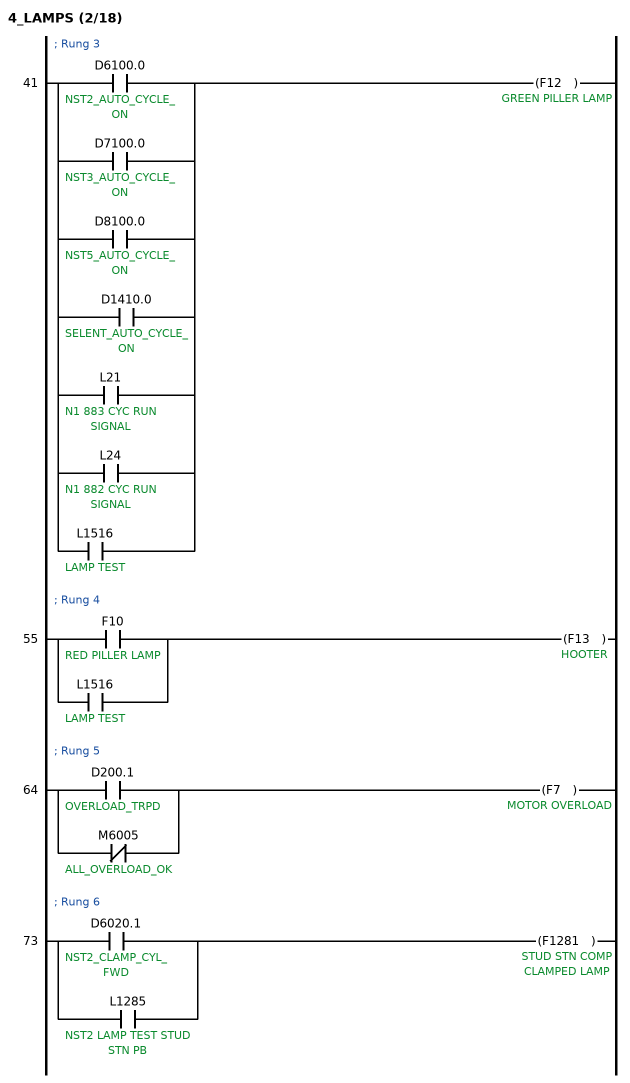
[picture p48: ladder of 4_LAMPS, rungs at steps 41 to 73]
; Rung 3
41    LD      D6100.0  ; NST2_AUTO_CYCLE_ON
      OR      D7100.0  ; NST3_AUTO_CYCLE_ON
      OR      D8100.0  ; NST5_AUTO_CYCLE_ON
      OR      D1410.0  ; SELENT_AUTO_CYCLE_ON
      OR      L21  ; N1 883 CYC RUN SIGNAL
      OR      L24  ; N1 882 CYC RUN SIGNAL
      OR      L1516  ; LAMP TEST
      OUT     F12  ; GREEN PILLER LAMP
; Rung 4
55    LD      F10  ; RED PILLER LAMP
      OR      L1516  ; LAMP TEST
      OUT     F13  ; HOOTER
; Rung 5
64    LD      D200.1  ; OVERLOAD_TRPD
      ORI     M6005  ; ALL_OVERLOAD_OK
      OUT     F7  ; MOTOR OVERLOAD
; Rung 6
73    LD      D6020.1  ; NST2_CLAMP_CYL_FWD
      OR      L1285  ; NST2 LAMP TEST STUD STN PB
      OUT     F1281  ; STUD STN COMP CLAMPED LAMP
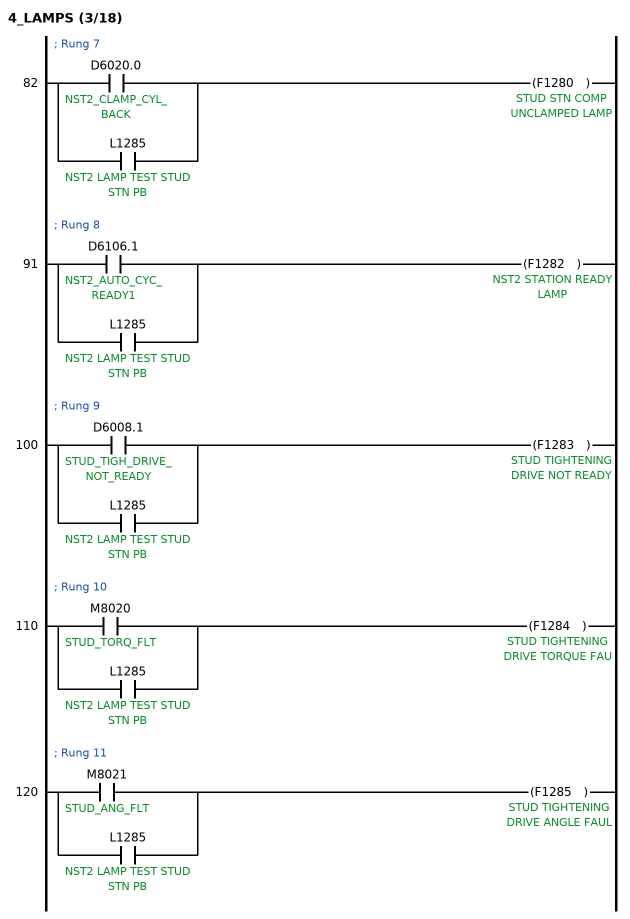
; Rung 7
82    LD      D6020.0  ; NST2_CLAMP_CYL_BACK
      OR      L1285  ; NST2 LAMP TEST STUD STN PB
      OUT     F1280  ; STUD STN COMP UNCLAMPED LAMP
; Rung 8
91    LD      D6106.1  ; NST2_AUTO_CYC_READY1
      OR      L1285  ; NST2 LAMP TEST STUD STN PB
      OUT     F1282  ; NST2 STATION READY LAMP
; Rung 9
100   LD      D6008.1  ; STUD_TIGH_DRIVE_NOT_READY
      OR      L1285  ; NST2 LAMP TEST STUD STN PB
      OUT     F1283  ; STUD TIGHTENING DRIVE NOT READY
; Rung 10
110   LD      M8020  ; STUD_TORQ_FLT
      OR      L1285  ; NST2 LAMP TEST STUD STN PB
      OUT     F1284  ; STUD TIGHTENING DRIVE TORQUE FAU
; Rung 11
120   LD      M8021  ; STUD_ANG_FLT
      OR      L1285  ; NST2 LAMP TEST STUD STN PB
      OUT     F1285  ; STUD TIGHTENING DRIVE ANGLE FAUL
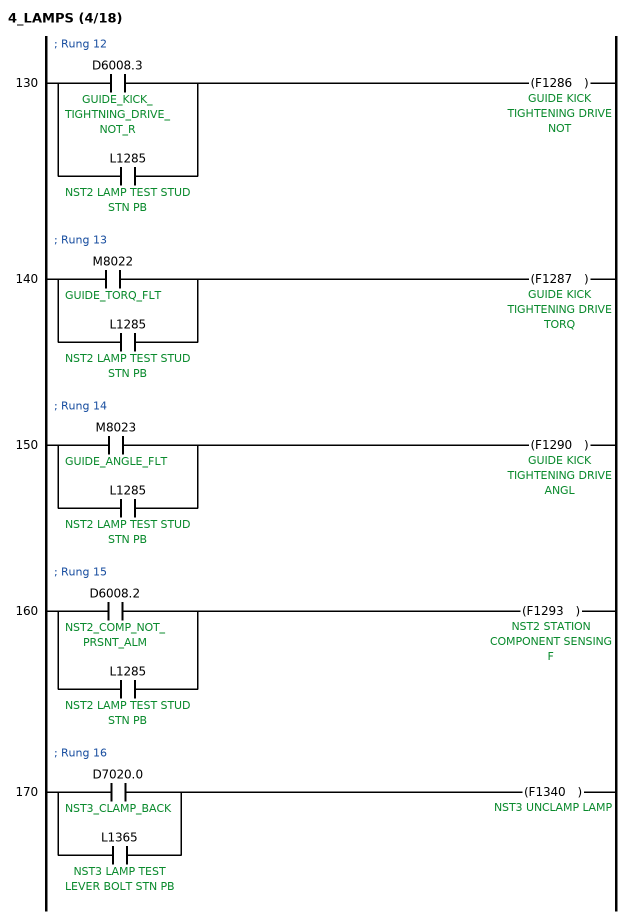
; Rung 12
130   LD      D6008.3  ; GUIDE_KICK_TIGHTNING_DRIVE_NOT_R
      OR      L1285  ; NST2 LAMP TEST STUD STN PB
      OUT     F1286  ; GUIDE KICK TIGHTENING DRIVE NOT
; Rung 13
140   LD      M8022  ; GUIDE_TORQ_FLT
      OR      L1285  ; NST2 LAMP TEST STUD STN PB
      OUT     F1287  ; GUIDE KICK TIGHTENING DRIVE TORQ
; Rung 14
150   LD      M8023  ; GUIDE_ANGLE_FLT
      OR      L1285  ; NST2 LAMP TEST STUD STN PB
      OUT     F1290  ; GUIDE KICK TIGHTENING DRIVE ANGL
; Rung 15
160   LD      D6008.2  ; NST2_COMP_NOT_PRSNT_ALM
      OR      L1285  ; NST2 LAMP TEST STUD STN PB
      OUT     F1293  ; NST2 STATION COMPONENT SENSING F
; Rung 16
170   LD      D7020.0  ; NST3_CLAMP_BACK
      OR      L1365  ; NST3 LAMP TEST LEVER BOLT STN PB
      OUT     F1340  ; NST3 UNCLAMP LAMP
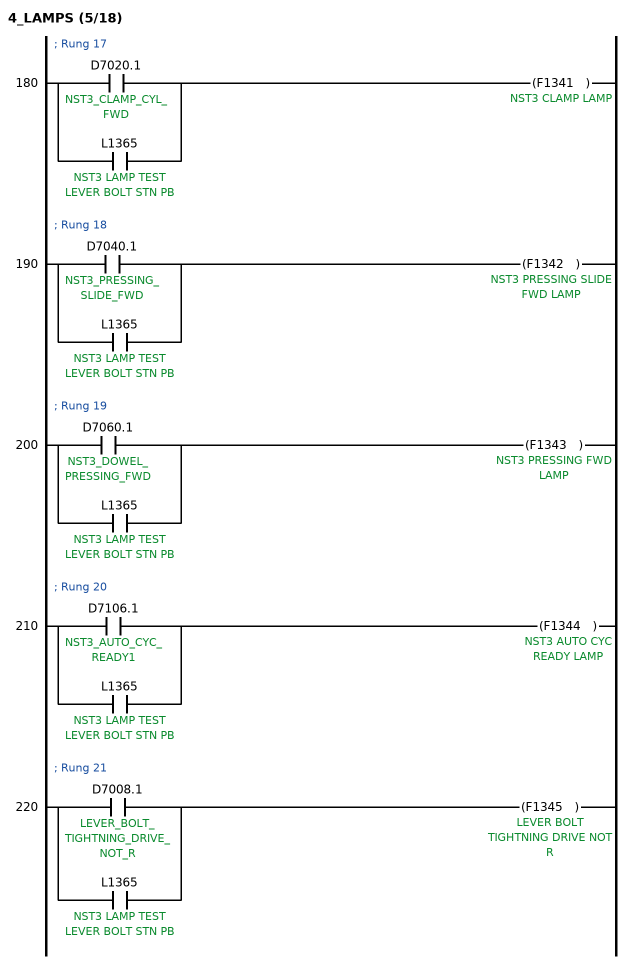
; Rung 17
180   LD      D7020.1  ; NST3_CLAMP_CYL_FWD
      OR      L1365  ; NST3 LAMP TEST LEVER BOLT STN PB
      OUT     F1341  ; NST3 CLAMP LAMP
; Rung 18
190   LD      D7040.1  ; NST3_PRESSING_SLIDE_FWD
      OR      L1365  ; NST3 LAMP TEST LEVER BOLT STN PB
      OUT     F1342  ; NST3 PRESSING SLIDE FWD LAMP
; Rung 19
200   LD      D7060.1  ; NST3_DOWEL_PRESSING_FWD
      OR      L1365  ; NST3 LAMP TEST LEVER BOLT STN PB
      OUT     F1343  ; NST3 PRESSING FWD LAMP
; Rung 20
210   LD      D7106.1  ; NST3_AUTO_CYC_READY1
      OR      L1365  ; NST3 LAMP TEST LEVER BOLT STN PB
      OUT     F1344  ; NST3 AUTO CYC READY LAMP
; Rung 21
220   LD      D7008.1  ; LEVER_BOLT_TIGHTNING_DRIVE_NOT_R
      OR      L1365  ; NST3 LAMP TEST LEVER BOLT STN PB
      OUT     F1345  ; LEVER BOLT TIGHTNING DRIVE NOT R
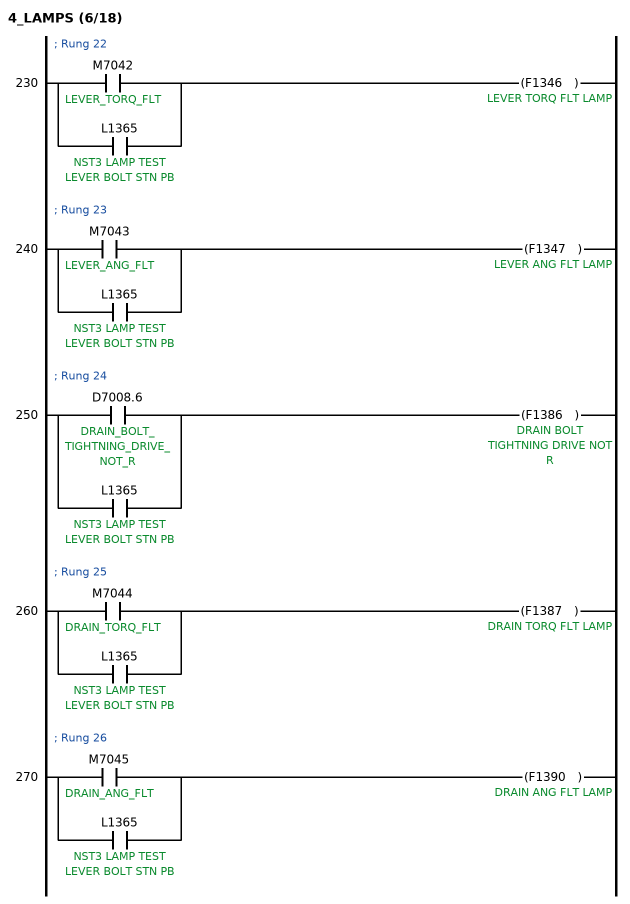
; Rung 22
230   LD      M7042  ; LEVER_TORQ_FLT
      OR      L1365  ; NST3 LAMP TEST LEVER BOLT STN PB
      OUT     F1346  ; LEVER TORQ FLT LAMP
; Rung 23
240   LD      M7043  ; LEVER_ANG_FLT
      OR      L1365  ; NST3 LAMP TEST LEVER BOLT STN PB
      OUT     F1347  ; LEVER ANG FLT LAMP
; Rung 24
250   LD      D7008.6  ; DRAIN_BOLT_TIGHTNING_DRIVE_NOT_R
      OR      L1365  ; NST3 LAMP TEST LEVER BOLT STN PB
      OUT     F1386  ; DRAIN BOLT TIGHTNING DRIVE NOT R
; Rung 25
260   LD      M7044  ; DRAIN_TORQ_FLT
      OR      L1365  ; NST3 LAMP TEST LEVER BOLT STN PB
      OUT     F1387  ; DRAIN TORQ FLT LAMP
; Rung 26
270   LD      M7045  ; DRAIN_ANG_FLT
      OR      L1365  ; NST3 LAMP TEST LEVER BOLT STN PB
      OUT     F1390  ; DRAIN ANG FLT LAMP
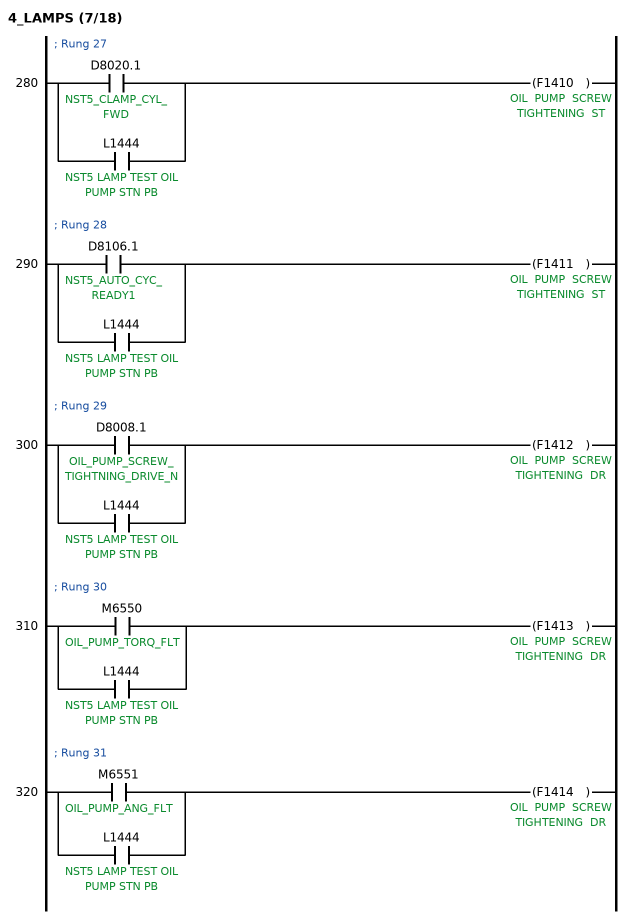
; Rung 27
280   LD      D8020.1  ; NST5_CLAMP_CYL_FWD
      OR      L1444  ; NST5 LAMP TEST OIL PUMP STN PB
      OUT     F1410  ; OIL  PUMP  SCREW  TIGHTENING  ST
; Rung 28
290   LD      D8106.1  ; NST5_AUTO_CYC_READY1
      OR      L1444  ; NST5 LAMP TEST OIL PUMP STN PB
      OUT     F1411  ; OIL  PUMP  SCREW  TIGHTENING  ST
; Rung 29
300   LD      D8008.1  ; OIL_PUMP_SCREW_TIGHTNING_DRIVE_N
      OR      L1444  ; NST5 LAMP TEST OIL PUMP STN PB
      OUT     F1412  ; OIL  PUMP  SCREW  TIGHTENING  DR
; Rung 30
310   LD      M6550  ; OIL_PUMP_TORQ_FLT
      OR      L1444  ; NST5 LAMP TEST OIL PUMP STN PB
      OUT     F1413  ; OIL  PUMP  SCREW  TIGHTENING  DR
; Rung 31
320   LD      M6551  ; OIL_PUMP_ANG_FLT
      OR      L1444  ; NST5 LAMP TEST OIL PUMP STN PB
      OUT     F1414  ; OIL  PUMP  SCREW  TIGHTENING  DR
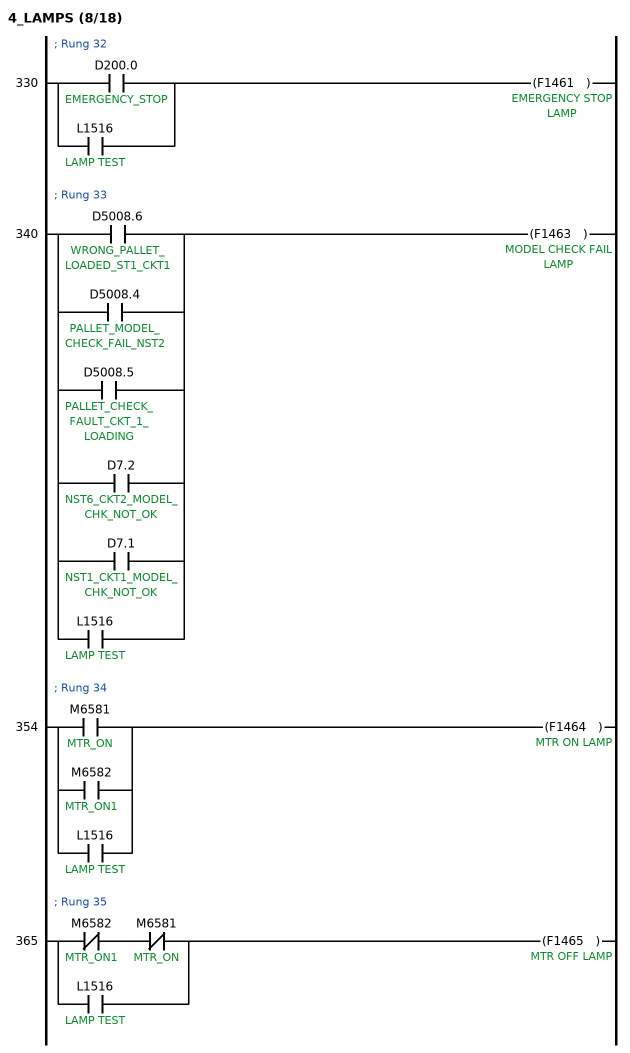
; Rung 32
330   LD      D200.0  ; EMERGENCY_STOP
      OR      L1516  ; LAMP TEST
      OUT     F1461  ; EMERGENCY STOP LAMP
; Rung 33
340   LD      D5008.6  ; WRONG_PALLET_LOADED_ST1_CKT1
      OR      D5008.4  ; PALLET_MODEL_CHECK_FAIL_NST2
      OR      D5008.5  ; PALLET_CHECK_FAULT_CKT_1_LOADING
      OR      D7.2  ; NST6_CKT2_MODEL_CHK_NOT_OK
      OR      D7.1  ; NST1_CKT1_MODEL_CHK_NOT_OK
      OR      L1516  ; LAMP TEST
      OUT     F1463  ; MODEL CHECK FAIL LAMP
; Rung 34
354   LD      M6581  ; MTR_ON
      OR      M6582  ; MTR_ON1
      OR      L1516  ; LAMP TEST
      OUT     F1464  ; MTR ON LAMP
; Rung 35
365   LDI     M6582  ; MTR_ON1
      ANI     M6581  ; MTR_ON
      OR      L1516  ; LAMP TEST
      OUT     F1465  ; MTR OFF LAMP
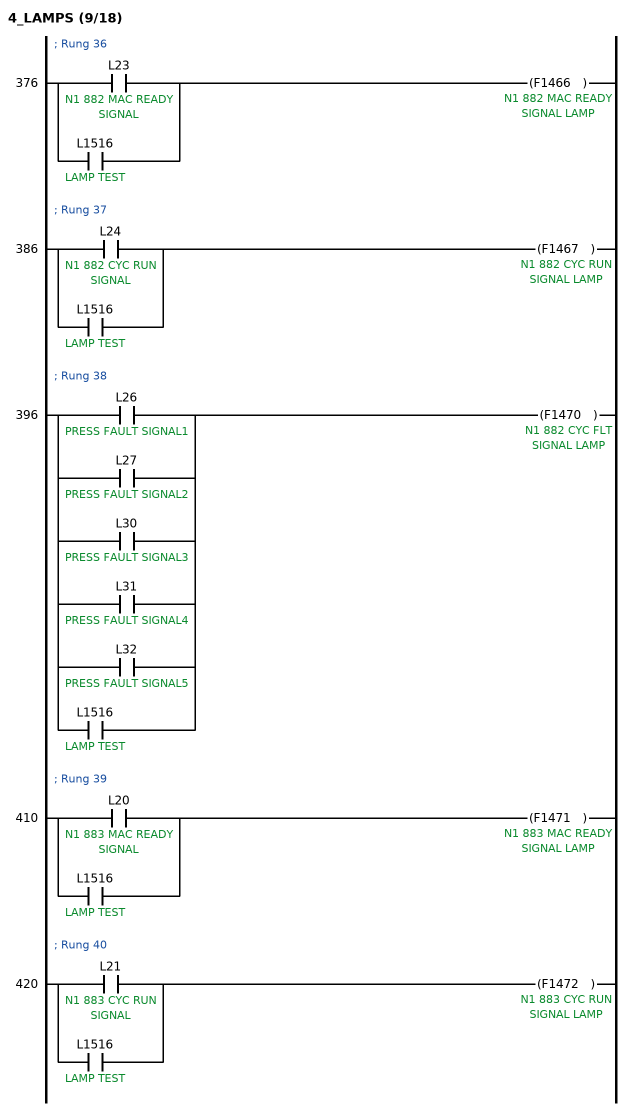
; Rung 36
376   LD      L23  ; N1 882 MAC READY SIGNAL
      OR      L1516  ; LAMP TEST
      OUT     F1466  ; N1 882 MAC READY SIGNAL LAMP
; Rung 37
386   LD      L24  ; N1 882 CYC RUN SIGNAL
      OR      L1516  ; LAMP TEST
      OUT     F1467  ; N1 882 CYC RUN SIGNAL LAMP
; Rung 38
396   LD      L26  ; PRESS FAULT SIGNAL1
      OR      L27  ; PRESS FAULT SIGNAL2
      OR      L30  ; PRESS FAULT SIGNAL3
      OR      L31  ; PRESS FAULT SIGNAL4
      OR      L32  ; PRESS FAULT SIGNAL5
      OR      L1516  ; LAMP TEST
      OUT     F1470  ; N1 882 CYC FLT SIGNAL LAMP
; Rung 39
410   LD      L20  ; N1 883 MAC READY SIGNAL
      OR      L1516  ; LAMP TEST
      OUT     F1471  ; N1 883 MAC READY SIGNAL LAMP
; Rung 40
420   LD      L21  ; N1 883 CYC RUN SIGNAL
      OR      L1516  ; LAMP TEST
      OUT     F1472  ; N1 883 CYC RUN SIGNAL LAMP
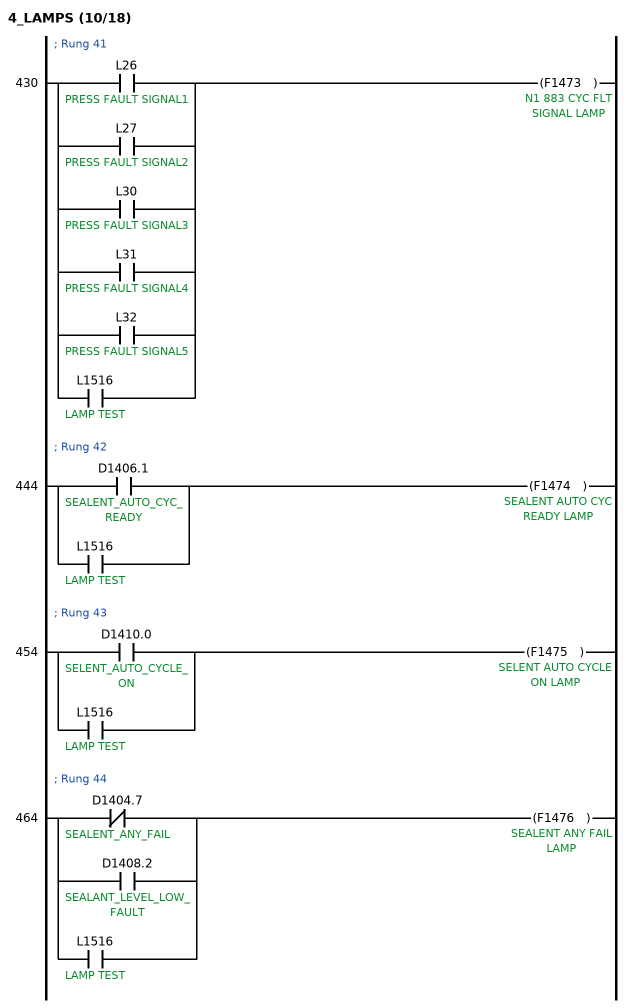
; Rung 41
430   LD      L26  ; PRESS FAULT SIGNAL1
      OR      L27  ; PRESS FAULT SIGNAL2
      OR      L30  ; PRESS FAULT SIGNAL3
      OR      L31  ; PRESS FAULT SIGNAL4
      OR      L32  ; PRESS FAULT SIGNAL5
      OR      L1516  ; LAMP TEST
      OUT     F1473  ; N1 883 CYC FLT SIGNAL LAMP
; Rung 42
444   LD      D1406.1  ; SEALENT_AUTO_CYC_READY
      OR      L1516  ; LAMP TEST
      OUT     F1474  ; SEALENT AUTO CYC READY LAMP
; Rung 43
454   LD      D1410.0  ; SELENT_AUTO_CYCLE_ON
      OR      L1516  ; LAMP TEST
      OUT     F1475  ; SELENT AUTO CYCLE ON LAMP
; Rung 44
464   LDI     D1404.7  ; SEALENT_ANY_FAIL
      OR      D1408.2  ; SEALANT_LEVEL_LOW_FAULT
      OR      L1516  ; LAMP TEST
      OUT     F1476  ; SEALENT ANY FAIL LAMP
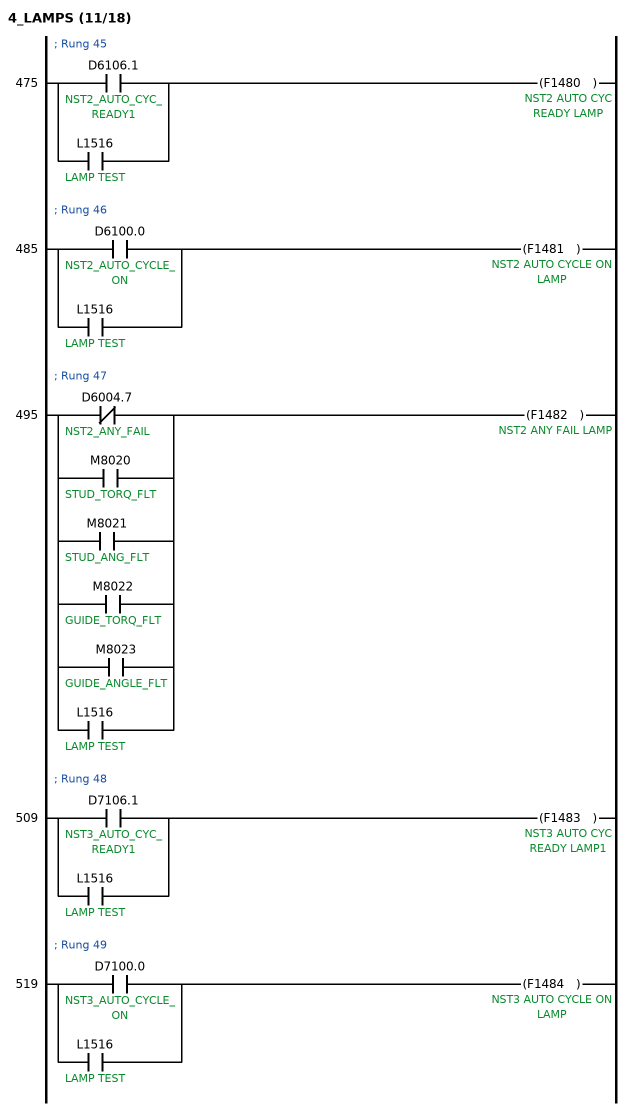
; Rung 45
475   LD      D6106.1  ; NST2_AUTO_CYC_READY1
      OR      L1516  ; LAMP TEST
      OUT     F1480  ; NST2 AUTO CYC READY LAMP
; Rung 46
485   LD      D6100.0  ; NST2_AUTO_CYCLE_ON
      OR      L1516  ; LAMP TEST
      OUT     F1481  ; NST2 AUTO CYCLE ON LAMP
; Rung 47
495   LDI     D6004.7  ; NST2_ANY_FAIL
      OR      M8020  ; STUD_TORQ_FLT
      OR      M8021  ; STUD_ANG_FLT
      OR      M8022  ; GUIDE_TORQ_FLT
      OR      M8023  ; GUIDE_ANGLE_FLT
      OR      L1516  ; LAMP TEST
      OUT     F1482  ; NST2 ANY FAIL LAMP
; Rung 48
509   LD      D7106.1  ; NST3_AUTO_CYC_READY1
      OR      L1516  ; LAMP TEST
      OUT     F1483  ; NST3 AUTO CYC READY LAMP1
; Rung 49
519   LD      D7100.0  ; NST3_AUTO_CYCLE_ON
      OR      L1516  ; LAMP TEST
      OUT     F1484  ; NST3 AUTO CYCLE ON LAMP
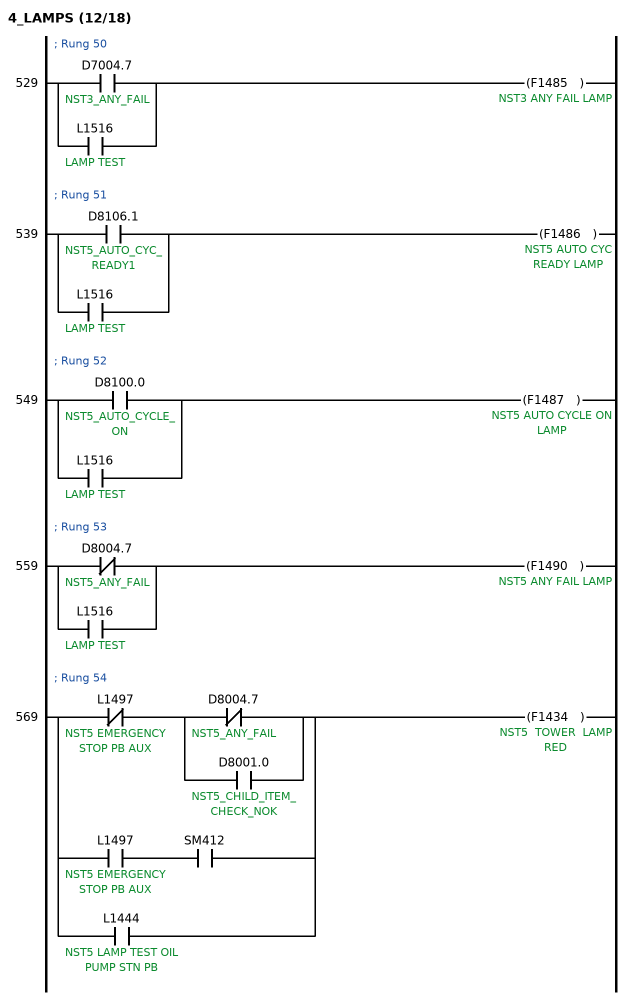
; Rung 50
529   LD      D7004.7  ; NST3_ANY_FAIL
      OR      L1516  ; LAMP TEST
      OUT     F1485  ; NST3 ANY FAIL LAMP
; Rung 51
539   LD      D8106.1  ; NST5_AUTO_CYC_READY1
      OR      L1516  ; LAMP TEST
      OUT     F1486  ; NST5 AUTO CYC READY LAMP
; Rung 52
549   LD      D8100.0  ; NST5_AUTO_CYCLE_ON
      OR      L1516  ; LAMP TEST
      OUT     F1487  ; NST5 AUTO CYCLE ON LAMP
; Rung 53
559   LDI     D8004.7  ; NST5_ANY_FAIL
      OR      L1516  ; LAMP TEST
      OUT     F1490  ; NST5 ANY FAIL LAMP
; Rung 54
569   LDI     L1497  ; NST5 EMERGENCY STOP PB AUX
      LDI     D8004.7  ; NST5_ANY_FAIL
      OR      D8001.0  ; NST5_CHILD_ITEM_CHECK_NOK
      ANB
      LD      L1497  ; NST5 EMERGENCY STOP PB AUX
      AND     SM412
      ORB
      OR      L1444  ; NST5 LAMP TEST OIL PUMP STN PB
      OUT     F1434  ; NST5  TOWER  LAMP  RED
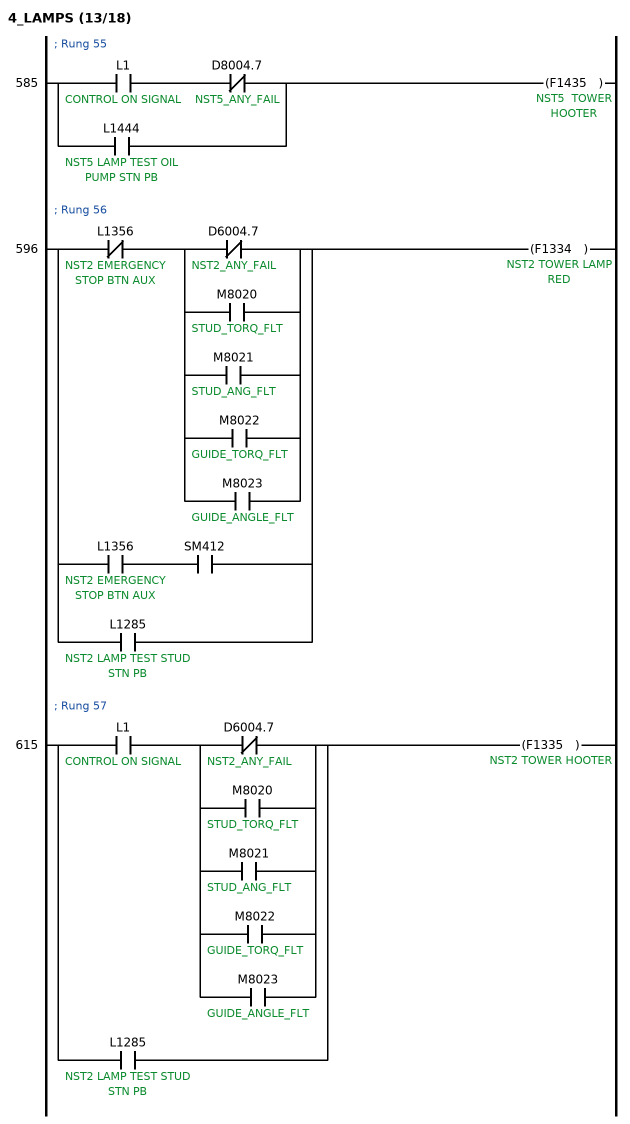
; Rung 55
585   LD      L1  ; CONTROL ON SIGNAL
      ANI     D8004.7  ; NST5_ANY_FAIL
      OR      L1444  ; NST5 LAMP TEST OIL PUMP STN PB
      OUT     F1435  ; NST5  TOWER  HOOTER
; Rung 56
596   LDI     L1356  ; NST2 EMERGENCY STOP BTN AUX
      LDI     D6004.7  ; NST2_ANY_FAIL
      OR      M8020  ; STUD_TORQ_FLT
      OR      M8021  ; STUD_ANG_FLT
      OR      M8022  ; GUIDE_TORQ_FLT
      OR      M8023  ; GUIDE_ANGLE_FLT
      ANB
      LD      L1356  ; NST2 EMERGENCY STOP BTN AUX
      AND     SM412
      ORB
      OR      L1285  ; NST2 LAMP TEST STUD STN PB
      OUT     F1334  ; NST2 TOWER LAMP RED
; Rung 57
615   LD      L1  ; CONTROL ON SIGNAL
      LDI     D6004.7  ; NST2_ANY_FAIL
      OR      M8020  ; STUD_TORQ_FLT
      OR      M8021  ; STUD_ANG_FLT
      OR      M8022  ; GUIDE_TORQ_FLT
      OR      M8023  ; GUIDE_ANGLE_FLT
      ANB
      OR      L1285  ; NST2 LAMP TEST STUD STN PB
      OUT     F1335  ; NST2 TOWER HOOTER
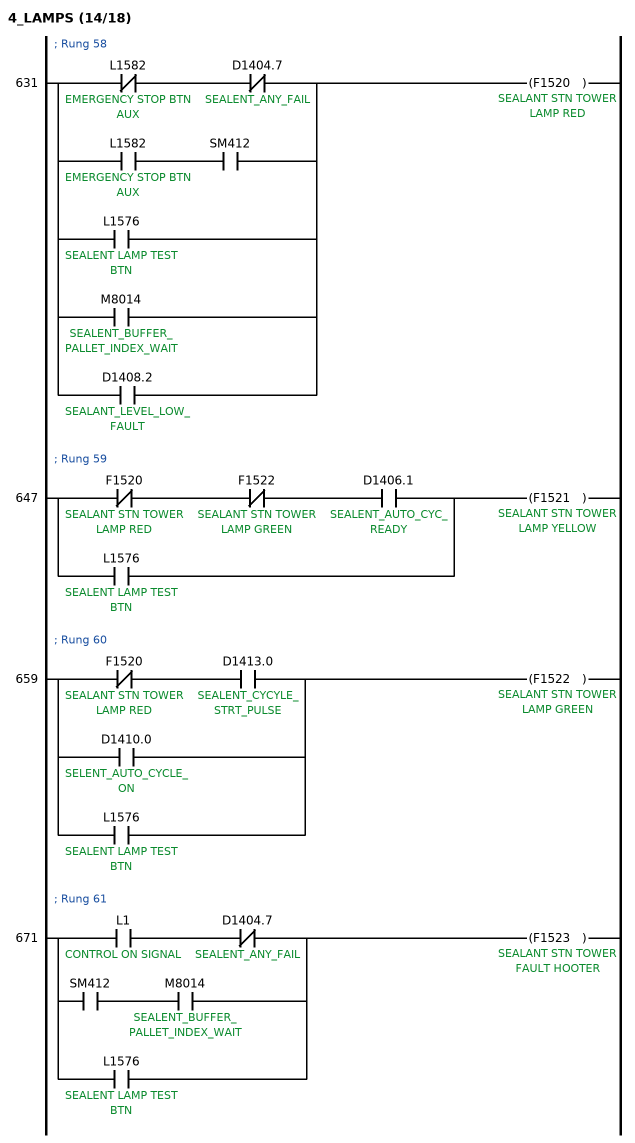
; Rung 58
631   LDI     L1582  ; EMERGENCY STOP BTN AUX
      ANI     D1404.7  ; SEALENT_ANY_FAIL
      LD      L1582  ; EMERGENCY STOP BTN AUX
      AND     SM412
      ORB
      OR      L1576  ; SEALENT LAMP TEST BTN
      OR      M8014  ; SEALENT_BUFFER_PALLET_INDEX_WAIT
      OR      D1408.2  ; SEALANT_LEVEL_LOW_FAULT
      OUT     F1520  ; SEALANT STN TOWER LAMP RED
; Rung 59
647   LDI     F1520  ; SEALANT STN TOWER LAMP RED
      ANI     F1522  ; SEALANT STN TOWER LAMP GREEN
      AND     D1406.1  ; SEALENT_AUTO_CYC_READY
      OR      L1576  ; SEALENT LAMP TEST BTN
      OUT     F1521  ; SEALANT STN TOWER LAMP YELLOW
; Rung 60
659   LDI     F1520  ; SEALANT STN TOWER LAMP RED
      AND     D1413.0  ; SEALENT_CYCYLE_STRT_PULSE
      OR      D1410.0  ; SELENT_AUTO_CYCLE_ON
      OR      L1576  ; SEALENT LAMP TEST BTN
      OUT     F1522  ; SEALANT STN TOWER LAMP GREEN
; Rung 61
671   LD      L1  ; CONTROL ON SIGNAL
      ANI     D1404.7  ; SEALENT_ANY_FAIL
      LD      SM412
      AND     M8014  ; SEALENT_BUFFER_PALLET_INDEX_WAIT
      ORB
      OR      L1576  ; SEALENT LAMP TEST BTN
      OUT     F1523  ; SEALANT STN TOWER FAULT HOOTER
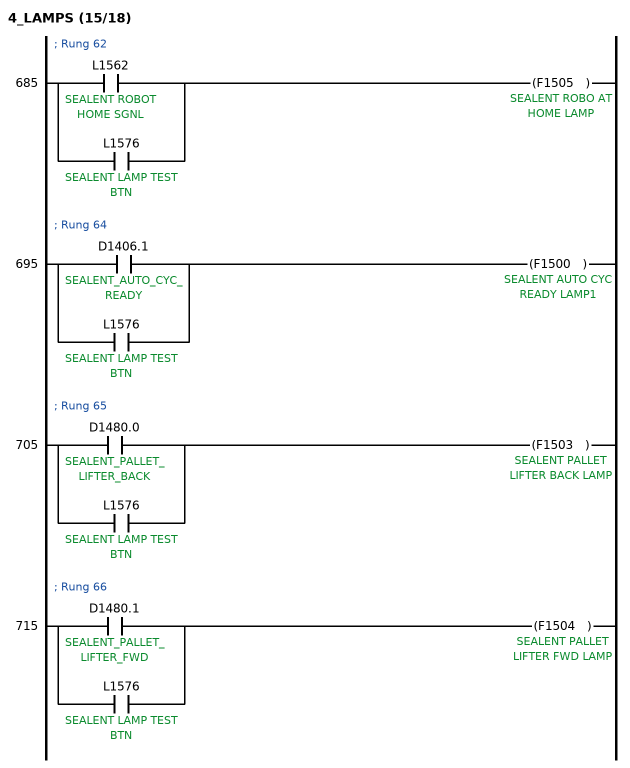
; Rung 62
685   LD      L1562  ; SEALENT ROBOT HOME SGNL
      OR      L1576  ; SEALENT LAMP TEST BTN
      OUT     F1505  ; SEALENT ROBO AT HOME LAMP
; Rung 64
695   LD      D1406.1  ; SEALENT_AUTO_CYC_READY
      OR      L1576  ; SEALENT LAMP TEST BTN
      OUT     F1500  ; SEALENT AUTO CYC READY LAMP1
; Rung 65
705   LD      D1480.0  ; SEALENT_PALLET_LIFTER_BACK
      OR      L1576  ; SEALENT LAMP TEST BTN
      OUT     F1503  ; SEALENT PALLET LIFTER BACK LAMP
; Rung 66
715   LD      D1480.1  ; SEALENT_PALLET_LIFTER_FWD
      OR      L1576  ; SEALENT LAMP TEST BTN
      OUT     F1504  ; SEALENT PALLET LIFTER FWD LAMP
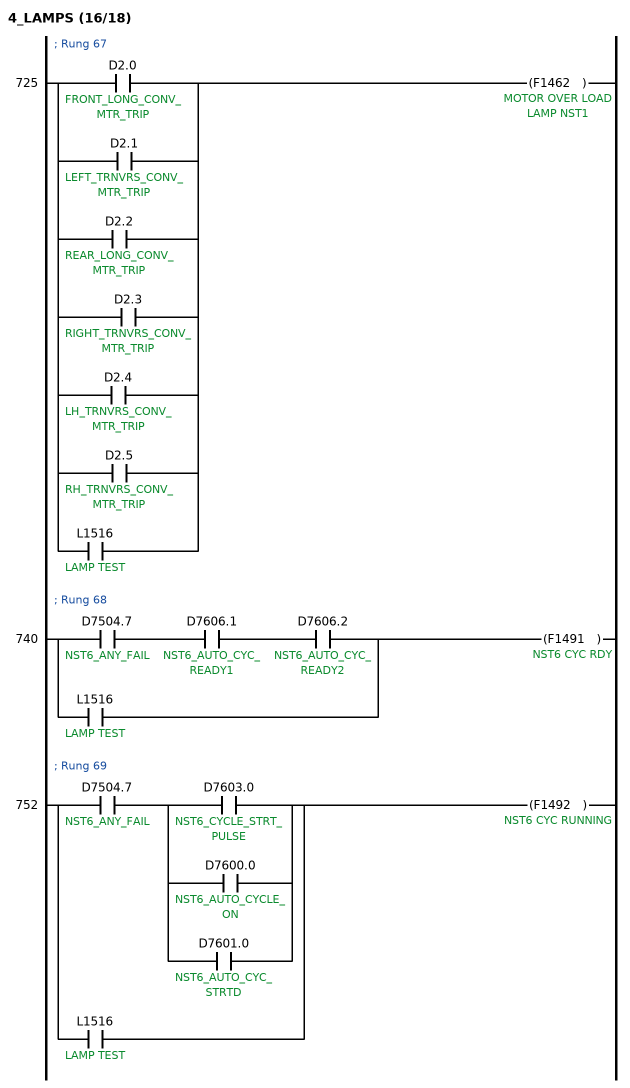
; Rung 67
725   LD      D2.0  ; FRONT_LONG_CONV_MTR_TRIP
      OR      D2.1  ; LEFT_TRNVRS_CONV_MTR_TRIP
      OR      D2.2  ; REAR_LONG_CONV_MTR_TRIP
      OR      D2.3  ; RIGHT_TRNVRS_CONV_MTR_TRIP
      OR      D2.4  ; LH_TRNVRS_CONV_MTR_TRIP
      OR      D2.5  ; RH_TRNVRS_CONV_MTR_TRIP
      OR      L1516  ; LAMP TEST
      OUT     F1462  ; MOTOR OVER LOAD LAMP NST1
; Rung 68
740   LD      D7504.7  ; NST6_ANY_FAIL
      AND     D7606.1  ; NST6_AUTO_CYC_READY1
      AND     D7606.2  ; NST6_AUTO_CYC_READY2
      OR      L1516  ; LAMP TEST
      OUT     F1491  ; NST6 CYC RDY
; Rung 69
752   LD      D7504.7  ; NST6_ANY_FAIL
      LD      D7603.0  ; NST6_CYCLE_STRT_PULSE
      OR      D7600.0  ; NST6_AUTO_CYCLE_ON
      OR      D7601.0  ; NST6_AUTO_CYC_STRTD
      ANB
      OR      L1516  ; LAMP TEST
      OUT     F1492  ; NST6 CYC RUNNING
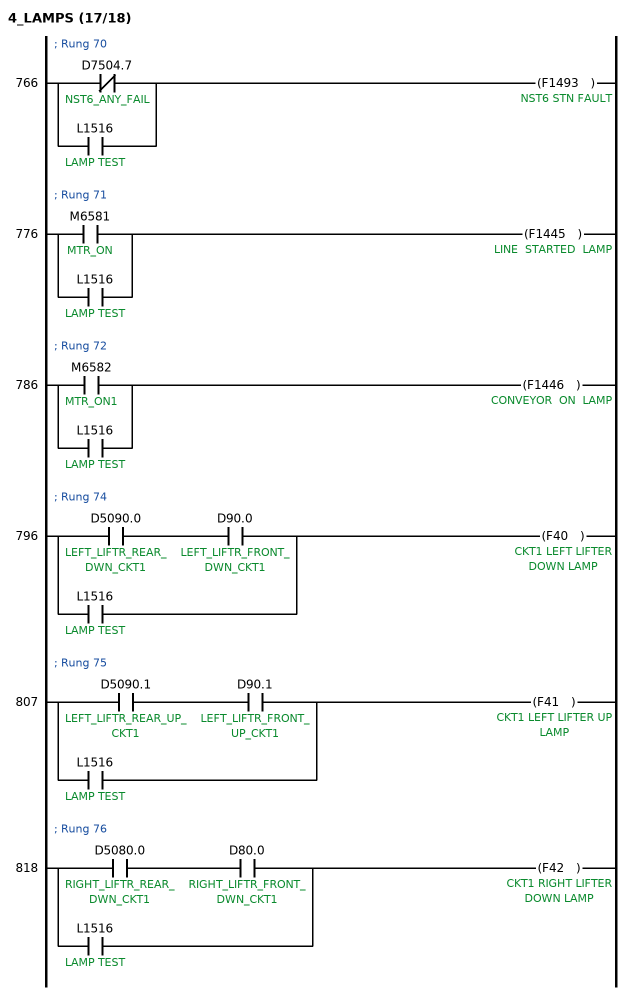
; Rung 70
766   LDI     D7504.7  ; NST6_ANY_FAIL
      OR      L1516  ; LAMP TEST
      OUT     F1493  ; NST6 STN FAULT
; Rung 71
776   LD      M6581  ; MTR_ON
      OR      L1516  ; LAMP TEST
      OUT     F1445  ; LINE  STARTED  LAMP
; Rung 72
786   LD      M6582  ; MTR_ON1
      OR      L1516  ; LAMP TEST
      OUT     F1446  ; CONVEYOR  ON  LAMP
; Rung 74
796   LD      D5090.0  ; LEFT_LIFTR_REAR_DWN_CKT1
      AND     D90.0  ; LEFT_LIFTR_FRONT_DWN_CKT1
      OR      L1516  ; LAMP TEST
      OUT     F40  ; CKT1 LEFT LIFTER DOWN LAMP
; Rung 75
807   LD      D5090.1  ; LEFT_LIFTR_REAR_UP_CKT1
      AND     D90.1  ; LEFT_LIFTR_FRONT_UP_CKT1
      OR      L1516  ; LAMP TEST
      OUT     F41  ; CKT1 LEFT LIFTER UP LAMP
; Rung 76
818   LD      D5080.0  ; RIGHT_LIFTR_REAR_DWN_CKT1
      AND     D80.0  ; RIGHT_LIFTR_FRONT_DWN_CKT1
      OR      L1516  ; LAMP TEST
      OUT     F42  ; CKT1 RIGHT LIFTER DOWN LAMP
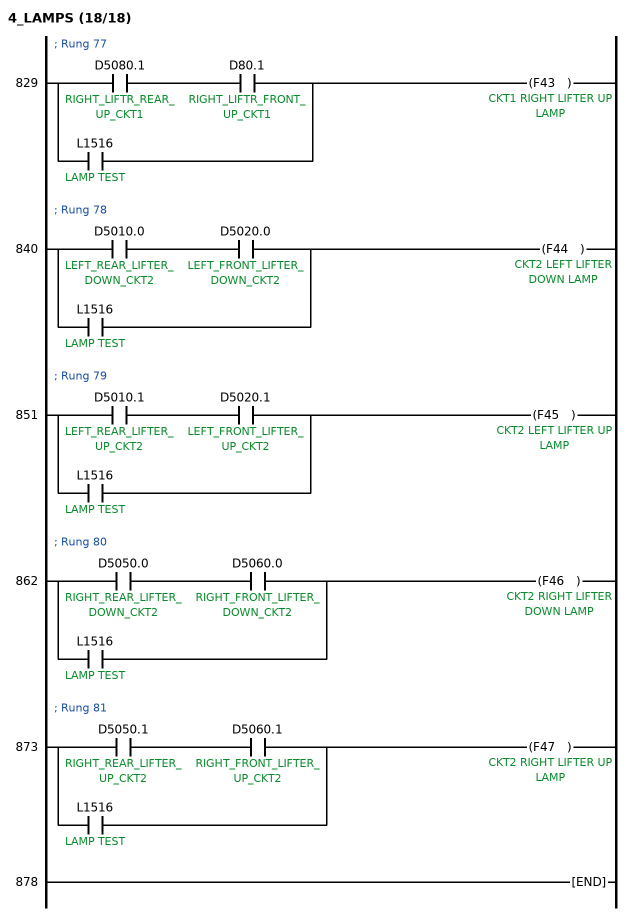
; Rung 77
829   LD      D5080.1  ; RIGHT_LIFTR_REAR_UP_CKT1
      AND     D80.1  ; RIGHT_LIFTR_FRONT_UP_CKT1
      OR      L1516  ; LAMP TEST
      OUT     F43  ; CKT1 RIGHT LIFTER UP LAMP
; Rung 78
840   LD      D5010.0  ; LEFT_REAR_LIFTER_DOWN_CKT2
      AND     D5020.0  ; LEFT_FRONT_LIFTER_DOWN_CKT2
      OR      L1516  ; LAMP TEST
      OUT     F44  ; CKT2 LEFT LIFTER DOWN LAMP
; Rung 79
851   LD      D5010.1  ; LEFT_REAR_LIFTER_UP_CKT2
      AND     D5020.1  ; LEFT_FRONT_LIFTER_UP_CKT2
      OR      L1516  ; LAMP TEST
      OUT     F45  ; CKT2 LEFT LIFTER UP LAMP
; Rung 80
862   LD      D5050.0  ; RIGHT_REAR_LIFTER_DOWN_CKT2
      AND     D5060.0  ; RIGHT_FRONT_LIFTER_DOWN_CKT2
      OR      L1516  ; LAMP TEST
      OUT     F46  ; CKT2 RIGHT LIFTER DOWN LAMP
; Rung 81
873   LD      D5050.1  ; RIGHT_REAR_LIFTER_UP_CKT2
      AND     D5060.1  ; RIGHT_FRONT_LIFTER_UP_CKT2
      OR      L1516  ; LAMP TEST
      OUT     F47  ; CKT2 RIGHT LIFTER UP LAMP
878   END
END_PROGRAM

PROGRAM 5_LEFT  // TRANSVERSE CKT1
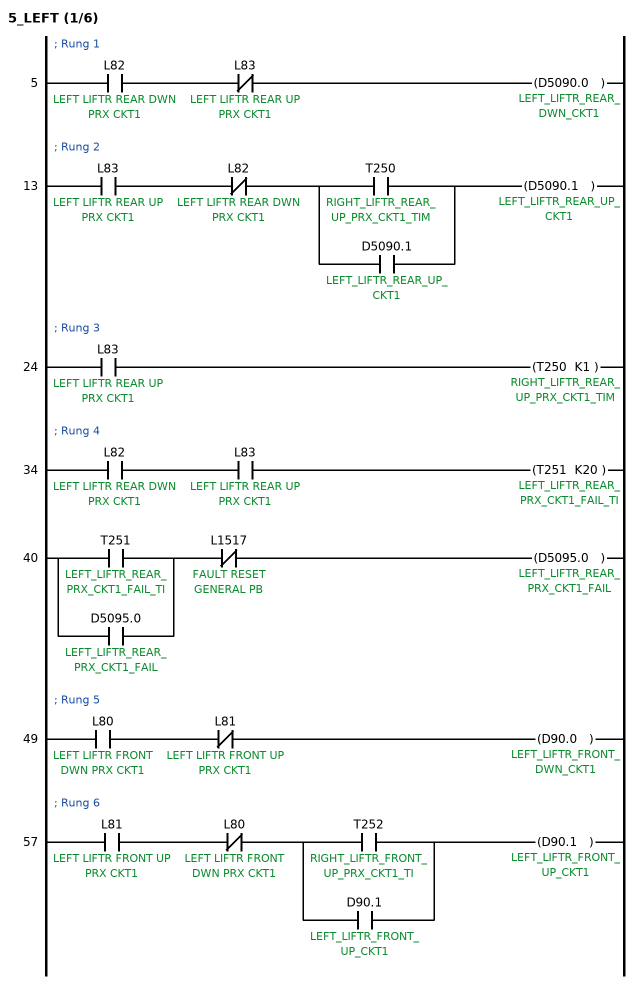
; Rung 1
5     LD      L82  ; LEFT LIFTR REAR DWN PRX CKT1
      ANI     L83  ; LEFT LIFTR REAR UP PRX CKT1
      OUT     D5090.0  ; LEFT_LIFTR_REAR_DWN_CKT1
; Rung 2
13    LD      L83  ; LEFT LIFTR REAR UP PRX CKT1
      ANI     L82  ; LEFT LIFTR REAR DWN PRX CKT1
      LD      T250  ; RIGHT_LIFTR_REAR_UP_PRX_CKT1_TIM
      OR      D5090.1  ; LEFT_LIFTR_REAR_UP_CKT1
      ANB
      OUT     D5090.1  ; LEFT_LIFTR_REAR_UP_CKT1
; Rung 3
24    LD      L83  ; LEFT LIFTR REAR UP PRX CKT1
      OUT     T250 K1  ; RIGHT_LIFTR_REAR_UP_PRX_CKT1_TIM
; Rung 4
34    LD      L82  ; LEFT LIFTR REAR DWN PRX CKT1
      AND     L83  ; LEFT LIFTR REAR UP PRX CKT1
      OUT     T251 K20  ; LEFT_LIFTR_REAR_PRX_CKT1_FAIL_TI
40    LD      T251  ; LEFT_LIFTR_REAR_PRX_CKT1_FAIL_TI
      OR      D5095.0  ; LEFT_LIFTR_REAR_PRX_CKT1_FAIL
      ANI     L1517  ; FAULT RESET GENERAL PB
      OUT     D5095.0  ; LEFT_LIFTR_REAR_PRX_CKT1_FAIL
; Rung 5
49    LD      L80  ; LEFT LIFTR FRONT DWN PRX CKT1
      ANI     L81  ; LEFT LIFTR FRONT UP PRX CKT1
      OUT     D90.0  ; LEFT_LIFTR_FRONT_DWN_CKT1
; Rung 6
57    LD      L81  ; LEFT LIFTR FRONT UP PRX CKT1
      ANI     L80  ; LEFT LIFTR FRONT DWN PRX CKT1
      LD      T252  ; RIGHT_LIFTR_FRONT_UP_PRX_CKT1_TI
      OR      D90.1  ; LEFT_LIFTR_FRONT_UP_CKT1
      ANB
      OUT     D90.1  ; LEFT_LIFTR_FRONT_UP_CKT1
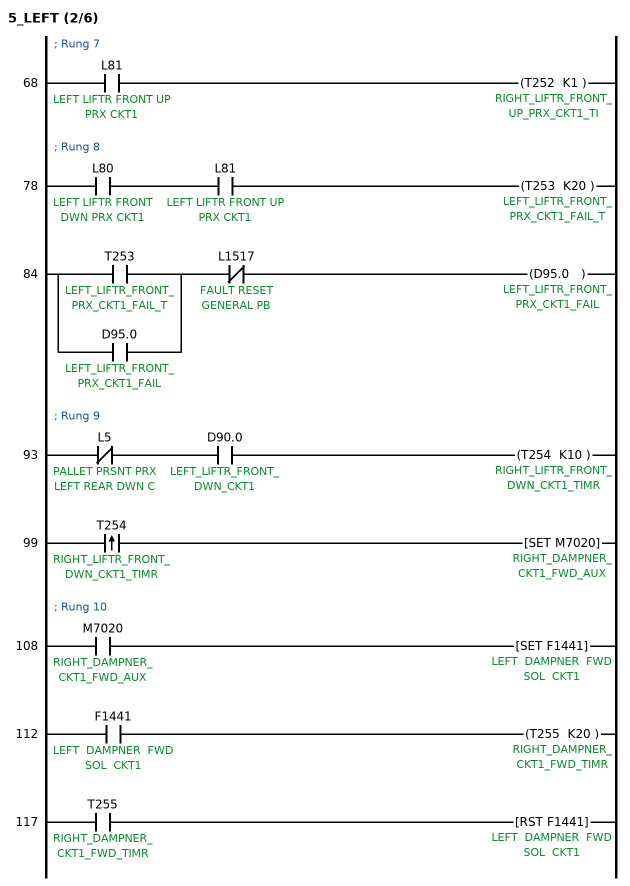
; Rung 7
68    LD      L81  ; LEFT LIFTR FRONT UP PRX CKT1
      OUT     T252 K1  ; RIGHT_LIFTR_FRONT_UP_PRX_CKT1_TI
; Rung 8
78    LD      L80  ; LEFT LIFTR FRONT DWN PRX CKT1
      AND     L81  ; LEFT LIFTR FRONT UP PRX CKT1
      OUT     T253 K20  ; LEFT_LIFTR_FRONT_PRX_CKT1_FAIL_T
84    LD      T253  ; LEFT_LIFTR_FRONT_PRX_CKT1_FAIL_T
      OR      D95.0  ; LEFT_LIFTR_FRONT_PRX_CKT1_FAIL
      ANI     L1517  ; FAULT RESET GENERAL PB
      OUT     D95.0  ; LEFT_LIFTR_FRONT_PRX_CKT1_FAIL
; Rung 9
93    LDI     L5  ; PALLET PRSNT PRX LEFT REAR DWN C
      AND     D90.0  ; LEFT_LIFTR_FRONT_DWN_CKT1
      OUT     T254 K10  ; RIGHT_LIFTR_FRONT_DWN_CKT1_TIMR
99    LDP     T254  ; RIGHT_LIFTR_FRONT_DWN_CKT1_TIMR
      SET     M7020  ; RIGHT_DAMPNER_CKT1_FWD_AUX
; Rung 10
108   LD      M7020  ; RIGHT_DAMPNER_CKT1_FWD_AUX
      SET     F1441  ; LEFT  DAMPNER  FWD  SOL  CKT1
112   LD      F1441  ; LEFT  DAMPNER  FWD  SOL  CKT1
      OUT     T255 K20  ; RIGHT_DAMPNER_CKT1_FWD_TIMR
117   LD      T255  ; RIGHT_DAMPNER_CKT1_FWD_TIMR
      RST     F1441  ; LEFT  DAMPNER  FWD  SOL  CKT1
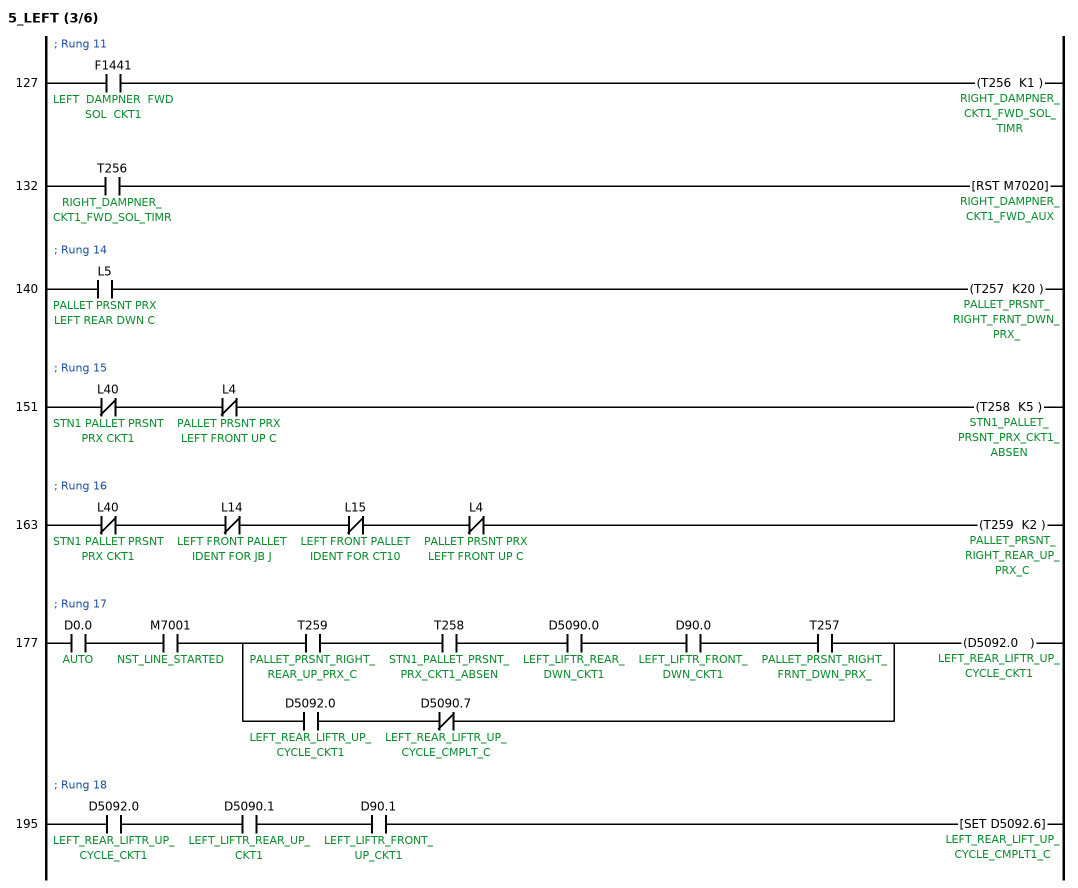
; Rung 11
127   LD      F1441  ; LEFT  DAMPNER  FWD  SOL  CKT1
      OUT     T256 K1  ; RIGHT_DAMPNER_CKT1_FWD_SOL_TIMR
132   LD      T256  ; RIGHT_DAMPNER_CKT1_FWD_SOL_TIMR
      RST     M7020  ; RIGHT_DAMPNER_CKT1_FWD_AUX
; Rung 14
140   LD      L5  ; PALLET PRSNT PRX LEFT REAR DWN C
      OUT     T257 K20  ; PALLET_PRSNT_RIGHT_FRNT_DWN_PRX_
; Rung 15
151   LDI     L40  ; STN1 PALLET PRSNT PRX CKT1
      ANI     L4  ; PALLET PRSNT PRX LEFT FRONT UP C
      OUT     T258 K5  ; STN1_PALLET_PRSNT_PRX_CKT1_ABSEN
; Rung 16
163   LDI     L40  ; STN1 PALLET PRSNT PRX CKT1
      ANI     L14  ; LEFT FRONT PALLET IDENT FOR JB J
      ANI     L15  ; LEFT FRONT PALLET IDENT FOR CT10
      ANI     L4  ; PALLET PRSNT PRX LEFT FRONT UP C
      OUT     T259 K2  ; PALLET_PRSNT_RIGHT_REAR_UP_PRX_C
; Rung 17
177   LD      D0.0  ; AUTO
      AND     M7001  ; NST_LINE_STARTED
      LD      T259  ; PALLET_PRSNT_RIGHT_REAR_UP_PRX_C
      AND     T258  ; STN1_PALLET_PRSNT_PRX_CKT1_ABSEN
      AND     D5090.0  ; LEFT_LIFTR_REAR_DWN_CKT1
      AND     D90.0  ; LEFT_LIFTR_FRONT_DWN_CKT1
      AND     T257  ; PALLET_PRSNT_RIGHT_FRNT_DWN_PRX_
      LD      D5092.0  ; LEFT_REAR_LIFTR_UP_CYCLE_CKT1
      ANI     D5090.7  ; LEFT_REAR_LIFTR_UP_CYCLE_CMPLT_C
      ORB
      ANB
      OUT     D5092.0  ; LEFT_REAR_LIFTR_UP_CYCLE_CKT1
; Rung 18
195   LD      D5092.0  ; LEFT_REAR_LIFTR_UP_CYCLE_CKT1
      AND     D5090.1  ; LEFT_LIFTR_REAR_UP_CKT1
      AND     D90.1  ; LEFT_LIFTR_FRONT_UP_CKT1
      SET     D5092.6  ; LEFT_REAR_LIFT_UP_CYCLE_CMPLT1_C
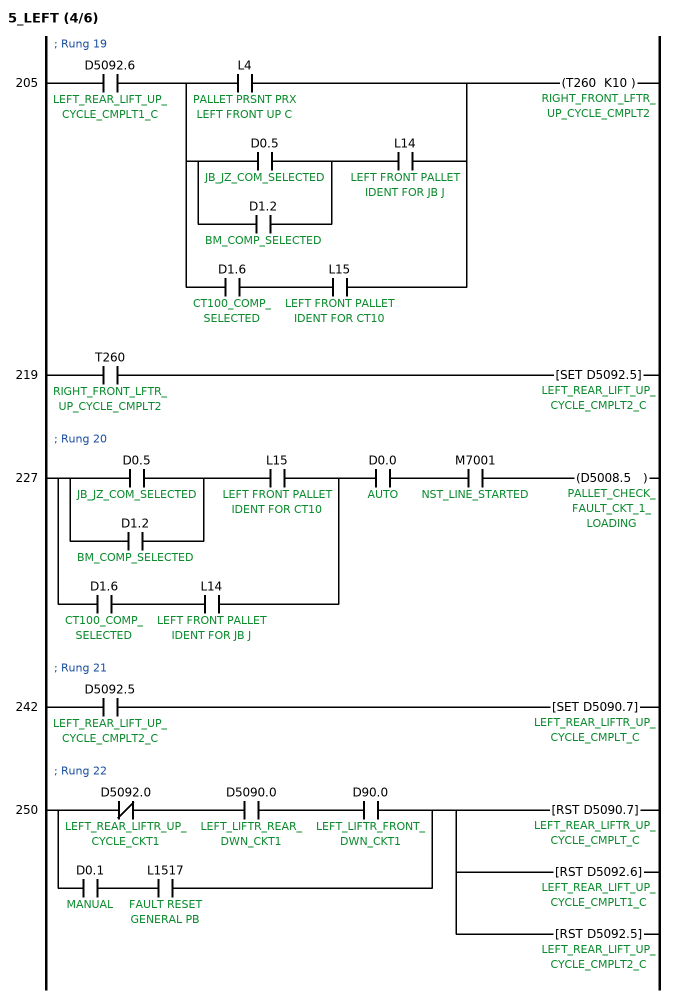
; Rung 19
205   LD      D5092.6  ; LEFT_REAR_LIFT_UP_CYCLE_CMPLT1_C
      LD      L4  ; PALLET PRSNT PRX LEFT FRONT UP C
      LD      D0.5  ; JB_JZ_COM_SELECTED
      OR      D1.2  ; BM_COMP_SELECTED
      AND     L14  ; LEFT FRONT PALLET IDENT FOR JB J
      ORB
      LD      D1.6  ; CT100_COMP_SELECTED
      AND     L15  ; LEFT FRONT PALLET IDENT FOR CT10
      ORB
      ANB
      OUT     T260 K10  ; RIGHT_FRONT_LFTR_UP_CYCLE_CMPLT2
219   LD      T260  ; RIGHT_FRONT_LFTR_UP_CYCLE_CMPLT2
      SET     D5092.5  ; LEFT_REAR_LIFT_UP_CYCLE_CMPLT2_C
; Rung 20
227   LD      D0.5  ; JB_JZ_COM_SELECTED
      OR      D1.2  ; BM_COMP_SELECTED
      AND     L15  ; LEFT FRONT PALLET IDENT FOR CT10
      LD      D1.6  ; CT100_COMP_SELECTED
      AND     L14  ; LEFT FRONT PALLET IDENT FOR JB J
      ORB
      AND     D0.0  ; AUTO
      AND     M7001  ; NST_LINE_STARTED
      OUT     D5008.5  ; PALLET_CHECK_FAULT_CKT_1_LOADING
; Rung 21
242   LD      D5092.5  ; LEFT_REAR_LIFT_UP_CYCLE_CMPLT2_C
      SET     D5090.7  ; LEFT_REAR_LIFTR_UP_CYCLE_CMPLT_C
; Rung 22
250   LDI     D5092.0  ; LEFT_REAR_LIFTR_UP_CYCLE_CKT1
      AND     D5090.0  ; LEFT_LIFTR_REAR_DWN_CKT1
      AND     D90.0  ; LEFT_LIFTR_FRONT_DWN_CKT1
      LD      D0.1  ; MANUAL
      AND     L1517  ; FAULT RESET GENERAL PB
      ORB
      RST     D5090.7  ; LEFT_REAR_LIFTR_UP_CYCLE_CMPLT_C
      RST     D5092.6  ; LEFT_REAR_LIFT_UP_CYCLE_CMPLT1_C
      RST     D5092.5  ; LEFT_REAR_LIFT_UP_CYCLE_CMPLT2_C
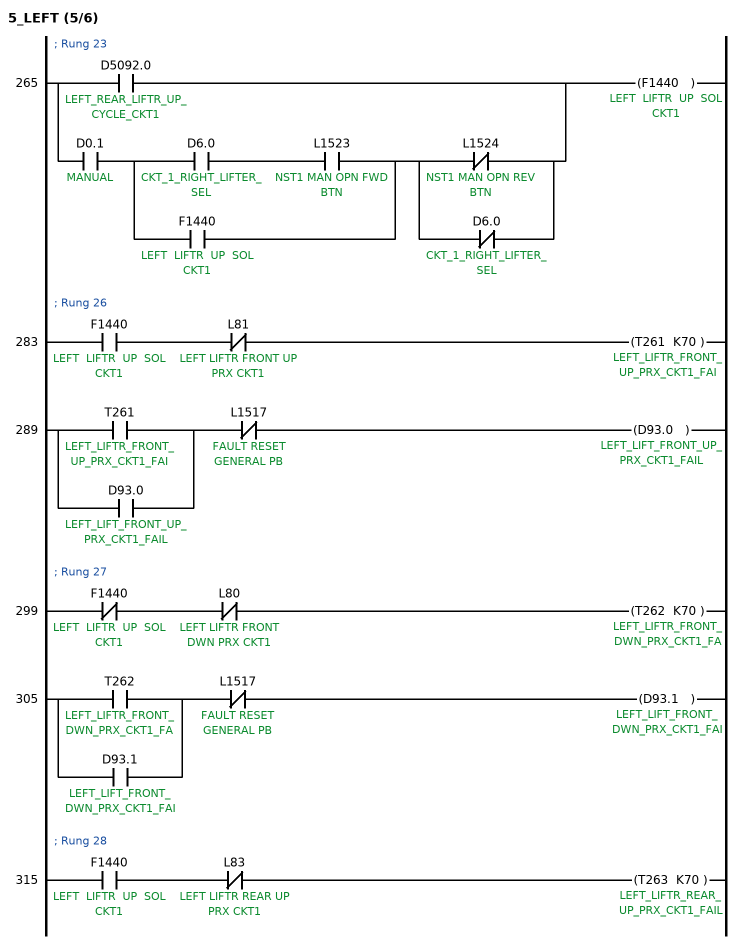
; Rung 23
265   LD      D5092.0  ; LEFT_REAR_LIFTR_UP_CYCLE_CKT1
      LD      D0.1  ; MANUAL
      LD      D6.0  ; CKT_1_RIGHT_LIFTER_SEL
      AND     L1523  ; NST1 MAN OPN FWD BTN
      OR      F1440  ; LEFT  LIFTR  UP  SOL  CKT1
      ANB
      LDI     L1524  ; NST1 MAN OPN REV BTN
      ORI     D6.0  ; CKT_1_RIGHT_LIFTER_SEL
      ANB
      ORB
      OUT     F1440  ; LEFT  LIFTR  UP  SOL  CKT1
; Rung 26
283   LD      F1440  ; LEFT  LIFTR  UP  SOL  CKT1
      ANI     L81  ; LEFT LIFTR FRONT UP PRX CKT1
      OUT     T261 K70  ; LEFT_LIFTR_FRONT_UP_PRX_CKT1_FAI
289   LD      T261  ; LEFT_LIFTR_FRONT_UP_PRX_CKT1_FAI
      OR      D93.0  ; LEFT_LIFT_FRONT_UP_PRX_CKT1_FAIL
      ANI     L1517  ; FAULT RESET GENERAL PB
      OUT     D93.0  ; LEFT_LIFT_FRONT_UP_PRX_CKT1_FAIL
; Rung 27
299   LDI     F1440  ; LEFT  LIFTR  UP  SOL  CKT1
      ANI     L80  ; LEFT LIFTR FRONT DWN PRX CKT1
      OUT     T262 K70  ; LEFT_LIFTR_FRONT_DWN_PRX_CKT1_FA
305   LD      T262  ; LEFT_LIFTR_FRONT_DWN_PRX_CKT1_FA
      OR      D93.1  ; LEFT_LIFT_FRONT_DWN_PRX_CKT1_FAI
      ANI     L1517  ; FAULT RESET GENERAL PB
      OUT     D93.1  ; LEFT_LIFT_FRONT_DWN_PRX_CKT1_FAI
; Rung 28
315   LD      F1440  ; LEFT  LIFTR  UP  SOL  CKT1
      ANI     L83  ; LEFT LIFTR REAR UP PRX CKT1
      OUT     T263 K70  ; LEFT_LIFTR_REAR_UP_PRX_CKT1_FAIL
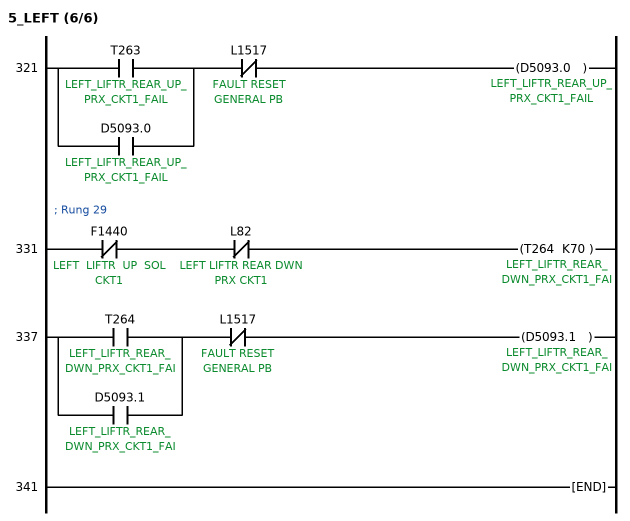
321   LD      T263  ; LEFT_LIFTR_REAR_UP_PRX_CKT1_FAIL
      OR      D5093.0  ; LEFT_LIFTR_REAR_UP_PRX_CKT1_FAIL
      ANI     L1517  ; FAULT RESET GENERAL PB
      OUT     D5093.0  ; LEFT_LIFTR_REAR_UP_PRX_CKT1_FAIL
; Rung 29
331   LDI     F1440  ; LEFT  LIFTR  UP  SOL  CKT1
      ANI     L82  ; LEFT LIFTR REAR DWN PRX CKT1
      OUT     T264 K70  ; LEFT_LIFTR_REAR_DWN_PRX_CKT1_FAI
337   LD      T264  ; LEFT_LIFTR_REAR_DWN_PRX_CKT1_FAI
      OR      D5093.1  ; LEFT_LIFTR_REAR_DWN_PRX_CKT1_FAI
      ANI     L1517  ; FAULT RESET GENERAL PB
      OUT     D5093.1  ; LEFT_LIFTR_REAR_DWN_PRX_CKT1_FAI
341   END
END_PROGRAM

PROGRAM 6_ALARM  // MAP
0     END
END_PROGRAM

PROGRAM 7_NEW  // ST1 CK2 
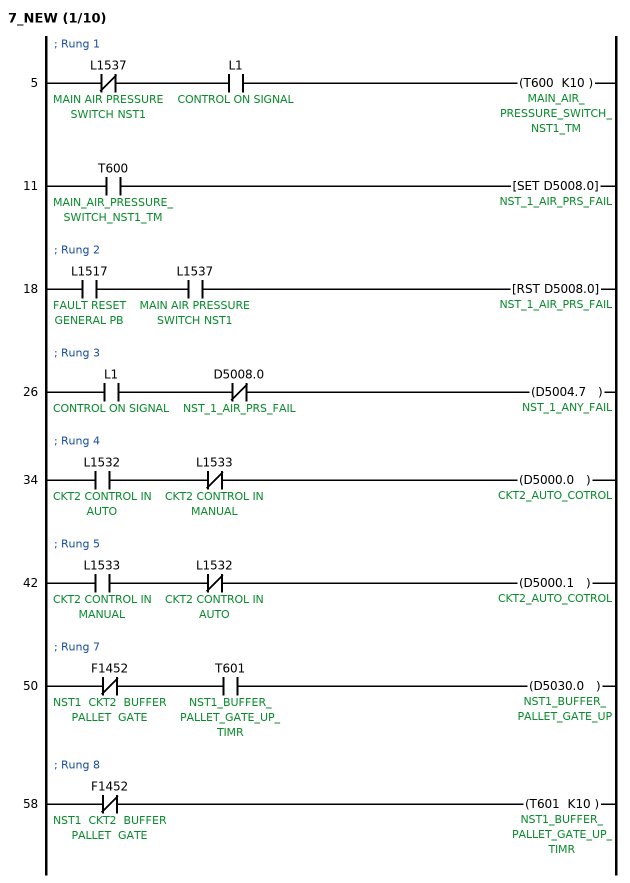
; Rung 1
5     LDI     L1537  ; MAIN AIR PRESSURE SWITCH NST1
      AND     L1  ; CONTROL ON SIGNAL
      OUT     T600 K10  ; MAIN_AIR_PRESSURE_SWITCH_NST1_TM
11    LD      T600  ; MAIN_AIR_PRESSURE_SWITCH_NST1_TM
      SET     D5008.0  ; NST_1_AIR_PRS_FAIL
; Rung 2
18    LD      L1517  ; FAULT RESET GENERAL PB
      AND     L1537  ; MAIN AIR PRESSURE SWITCH NST1
      RST     D5008.0  ; NST_1_AIR_PRS_FAIL
; Rung 3
26    LD      L1  ; CONTROL ON SIGNAL
      ANI     D5008.0  ; NST_1_AIR_PRS_FAIL
      OUT     D5004.7  ; NST_1_ANY_FAIL
; Rung 4
34    LD      L1532  ; CKT2 CONTROL IN AUTO
      ANI     L1533  ; CKT2 CONTROL IN MANUAL
      OUT     D5000.0  ; CKT2_AUTO_COTROL
; Rung 5
42    LD      L1533  ; CKT2 CONTROL IN MANUAL
      ANI     L1532  ; CKT2 CONTROL IN AUTO
      OUT     D5000.1  ; CKT2_AUTO_COTROL
; Rung 7
50    LDI     F1452  ; NST1  CKT2  BUFFER  PALLET  GATE
      AND     T601  ; NST1_BUFFER_PALLET_GATE_UP_TIMR
      OUT     D5030.0  ; NST1_BUFFER_PALLET_GATE_UP
; Rung 8
58    LDI     F1452  ; NST1  CKT2  BUFFER  PALLET  GATE
      OUT     T601 K10  ; NST1_BUFFER_PALLET_GATE_UP_TIMR
